TYPE ST_Supervisor :
	STRUCT
		DATA	: STRING;
		ERROR	: STRING;
	END_STRUCT
END_TYPE

(* stored: Version 1.1.0.1, ProductVersion 3.1.4026.18
   DUT ST_Supervisor: Id {2599c589-7966-412e-9002-2862bc44aefa} *)
